Staubli VAL3: isInLimits.pgx

program IsInLimits(bool& ret)
  local pointRx pt
  local bool err_x
  local bool err_y
  local bool err_z
begin
//*******************************************************************************
//*   ______
//*  / _____) /|
//* | |      / /
//* | | /\  / /
//* | | \ \/ /  _      Copyright (c) KEOLABS, 2016
//* | |  \__/  | |        http://www.keolabs.com
//* | |________| |
//*  \__________/
//*
//********************************************************************************
//*@file          : IsInLimits
//*@author        : Yves Ragot
//*@version       : $Id: isInLimits.pgx 1558 2017-01-05 08:13:36Z yves $
//*@brief         : Check the if the current position is in the limits
//*
//*******************************************************************************/

  // get current position
  pt = here(tCurrentTool, fCurrentFrame)

  // round values before comparing with limits (integer values)
  pt.trsf.x = round(pt.trsf.x * 10) / 10
  pt.trsf.y = round(pt.trsf.y * 10) / 10
  pt.trsf.z = round(pt.trsf.z * 10) / 10

  // check fatal limits
  err_x = (pt.trsf.x < CurLimitsTable["Xmin"]) or (pt.trsf.x > CurLimitsTable["Xmax"])
  err_y = (pt.trsf.y < CurLimitsTable["Ymin"]) or (pt.trsf.y > CurLimitsTable["Ymax"])
  err_z = (pt.trsf.z < CurLimitsTable["Zmin"]) or (pt.trsf.z > CurLimitsTable["Zmax"])

  // ret = true if position is correctly in limits
  ret = !(err_x or err_y or err_z)

end
